// TIA Portal V19 export
TYPE "typePressureGuageRs485Configuration"
TITLE = LBC_typeAnalogOutputConfiguration
// Module related configuration parameters
// stored: Access Published
   STRUCT
      referenceDesignator { S7_SetPoint := 'True'} : WString[25] := WSTRING#'AnalogOutput';   // Device name or device ID
      physicalUnit { S7_SetPoint := 'True'} : String[10] := 'unit';   // Each value should have a physical unit (like [°C], [kWh], etc.)
      isUnipolarSignal { S7_SetPoint := 'True'} : Bool := TRUE;   // TRUE: Sensor is a unipolar type (just positive values), FALSE: Sensor is a bipolar type (positive and negative values)
      default { S7_SetPoint := 'True'} : Int := 0;   // Default OUTPUT analog value to be returned if function block is not enabled or quality is bad
      limitHigh2 { S7_SetPoint := 'True'} : LReal := 90.0;   // Process value limit high 2
      limitHigh1 { S7_SetPoint := 'True'} : LReal := 80.0;   // Process value limit high 1
      limitLow1 { S7_SetPoint := 'True'} : LReal := -80.0;   // Process value limit low 1
      limitLow2 { S7_SetPoint := 'True'} : LReal := -90.0;   // Process value limit low 2
      processValueMax { S7_SetPoint := 'True'} : LReal := 100.0;   // Maximum limit of the process value
      processValueMin { S7_SetPoint := 'True'} : LReal := -100.0;   // Minimum limit of the process value
      scaleProcessUppPoint { S7_SetPoint := 'True'} : LReal := 100.0;   // Upper point for the process value
      scaleProcessLowPoint { S7_SetPoint := 'True'} : LReal := -100.0;   // Lower point for the process value
      scaleAnalogUppPoint { S7_SetPoint := 'True'} : LReal := 27648.0;   // Upper point for the analog output. Maximum value from the hardware module - i.e. 27648 - scaled value
      scaleAnalogLowPoint { S7_SetPoint := 'True'} : LReal := 0.0;   // Lower point for the analog output. Minimum value from the hardware module - i.e. 0 - scaled value
      disableAlarms { S7_SetPoint := 'True'} : Bool;   // Disable the alarms of the block
   END_STRUCT;
END_TYPE
